// TIA Portal V19 export
TYPE "UDT_STATUS_CVLV"
   STRUCT
      running : Bool;
      justStarted : Bool;
      justStopped : Bool;
      reference : Real;
      enabled { ExternalAccessible := 'False'; ExternalVisible := 'False'; ExternalWritable := 'False'} : Bool;
      old : Struct
         running : Bool;
      END_STRUCT;
   END_STRUCT;
END_TYPE
